FUNCTION_BLOCK TermFuse
VAR
	_input : BOOL;
	
END_VAR

PROPERTY IsActive : BOOL
GET
IsActive := _input;
END_GET
SET
_input := IsActive;
END_SET
END_PROPERTY

END_FUNCTION_BLOCK

(* stored: Version 1.1.0.1, ProductVersion 3.1.4024.12
   POU TermFuse: Id {a8875299-77d1-432d-981b-82ec5782068f}, SpecialFunc None
   Property IsActive: Id {c9d06f43-a262-42a7-97fc-e7cefa25fa55}
   Get Get: Id {55ae8ec7-bb02-45c6-95f9-60dab7c2bc54}
   Set Set: Id {ed525197-c64e-4ae9-88ee-a4f5f6af8c7d} *)
